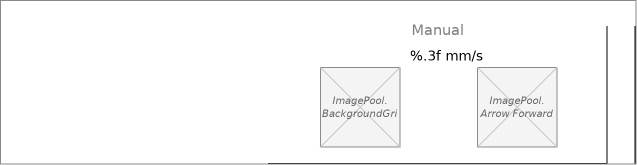
VISUALIZATION VisuAxisControl_1  // 637x165, background image ImagePool.BackgrounFrame
VAR_IN_OUT
	sAxisName_1		: STRING;
	stAxisVisu_1	: ST_AxisInterface;
END_VAR
    Line (635,163) (635,26), invisible if: PRG_Process.bInvisible
    Ellipse (333,77 52x55), invisible if: not stAxisVisu_1.In.xJogBw
    Image (320,67 80x80), image: ImagePool.BackgroundGri
    Ellipse (490,78 52x55), invisible if: not stAxisVisu_1.In.xJogFw
    Image (477,67 80x80), image: ImagePool.Arrow Forward
    Label (374,10 132x40), "Manual"
    Rectangle (389,42 97x28), "%.3f mm/s", text variable: stAxisVisu_1.In.fJogVelo
        OnMouseClick: write the text variable via VisuDialogs.Numpad
    Line (268,163) (607,163)
    InvisibleInput (323,67 86x78)
        tap stAxisVisu_1.In.xJogBw
    InvisibleInput (478,68 81x76)
        tap stAxisVisu_1.In.xJogFw
    Line (607,163) (607,26)
END_VISUALIZATION

(* stored: Version 1.1.0.1, ProductVersion 3.1.4022.6
   Visu VisuAxisControl_1: Id {caf945db-461b-427d-9de1-3dc9c68840d9} *)
